TYPE ST_BA_MyWeatherData :
STRUCT
	fWeatherTemperature		: REAL;
	fHumidity				: REAL;
	fBrightness				: REAL;
	fWindSpeed				: REAL;
	fWindDirection			: REAL;
	fLatitude				: REAL;
	fLongitude				: REAL;
	
	bDisturb				: BOOL;
END_STRUCT
END_TYPE

(* stored: Version 1.1.0.1, ProductVersion 3.1.4024.5
   DUT ST_BA_MyWeatherData: Id {c5fa38e3-4da4-4115-8cb6-d187ecff71f2} *)
